FUNCTION_BLOCK JSON_FORMER (* Basic FB with empty ECC *)
  (* Standard: 61499-2 *)
  (* Version 1.0, 2023-04-20, valentinnodan *)
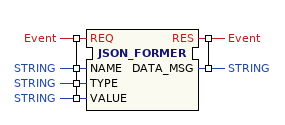
  EVENT_INPUT
    REQ WITH NAME, TYPE, VALUE;
  END_EVENT
  EVENT_OUTPUT
    RES WITH DATA_MSG;
  END_EVENT
  VAR_INPUT
    NAME : STRING;
    TYPE : STRING;
    VALUE : STRING;
  END_VAR
  VAR_OUTPUT
    DATA_MSG : STRING;
  END_VAR
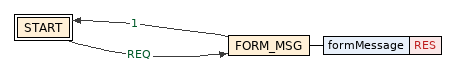
  EC_STATES
    START; (* Initial State *)
    FORM_MSG : formMessage -> RES;
  END_STATES
  EC_TRANSITIONS
    START TO FORM_MSG := REQ;
    FORM_MSG TO START := 1;
  END_TRANSITIONS
  ALGORITHM formMessage IN ST:
VAR
	openBrace: STRING;
	closeBrace: STRING;
	quote: STRING;
	splitter: STRING;
	separator: STRING;
	nameMsg:STRING;
	typeMsg: STRING;
	valueMsg: STRING;
	valueName: STRING;
	nameName: STRING;
	typeName: STRING;
END_VAR;
quote := '"';
openBrace := '{';
closeBrace := '}';
splitter:= ':';
separator:=',';
nameName:='NAME';
typeName:='TYPE';
valueName:='VALUE';
nameMsg:=CONCAT(quote, nameName, quote, splitter, quote, NAME, quote);
typeMsg:=CONCAT(quote, typeName, quote, splitter, quote, TYPE, quote);
valueMsg:=CONCAT(quote, valueName, quote, splitter, quote, VALUE, quote);
DATA_MSG:=CONCAT(CONCAT(openBrace, CONCAT(nameMsg, separator)), CONCAT(CONCAT(typeMsg, separator), CONCAT(valueMsg, closeBrace)));
  END_ALGORITHM
END_FUNCTION_BLOCK
